(* PLC project prj, KAIST_DSLAB noNameNow 1, author bwkim *)
(* stored: creationDateTime 2017-1-22T00:06:53, modificationDateTime 2017-1-22T00:06:55 *)

PROGRAM Program1____sub1
  VAR
    SELECTION : INT;
  END_VAR
  VAR_INPUT
    CLKIO_ABOX_UAIF0 : INT;
  END_VAR
  VAR_INPUT
    CLKIO_ABOX_UAIF1 : INT;
  END_VAR
  VAR_INPUT
    CLKIO_ABOX_UAIF2 : INT;
  END_VAR
  VAR_INPUT
    CLKIO_ABOX_UAIF3 : INT;
  END_VAR
  VAR_INPUT
    CLKIO_ABoX_UAIF4 : INT;
  END_VAR
  VAR_INPUT
    FIN : INT;
  END_VAR
  VAR_INPUT
    FINN : INT;
  END_VAR
  VAR_INPUT
    OSCCLK_ABOX : INT;
  END_VAR
  VAR_OUTPUT
    ABOX_DAR : INT;
  END_VAR
  VAR_OUTPUT
    ACLKM_BTM_ABOX : INT;
  END_VAR
  VAR_OUTPUT
    ACLKS_PERI_AXI_AS : INT;
  END_VAR
  VAR_OUTPUT
    ACLK_ABOX_TOP : INT;
  END_VAR
  VAR_OUTPUT
    ACLK_PMU_ABOX : INT;
  END_VAR
  VAR_OUTPUT
    ACLK_PPMU_ABOX : INT;
  END_VAR
  VAR_OUTPUT
    ACLK_SYSREG_ABOX : INT;
  END_VAR
  VAR_OUTPUT
    AUD_CODEC_MCLK_DFTMUX_ABOX : INT;
  END_VAR
  VAR_OUTPUT
    BCLK_DSIF_ABOX_TOP : INT;
  END_VAR
  VAR_OUTPUT
    BCLK_UAIF2_ABOX_TOP : INT;
  END_VAR
  VAR_OUTPUT
    BCLK_UAIF3_ABOX_TOP : INT;
  END_VAR
  VAR_OUTPUT
    BCLK_UAIF4_ABOX_TOP : INT;
  END_VAR
  VAR_OUTPUT
    BCLK_UAIF_ABOX_TOP : INT;
  END_VAR
  VAR_OUTPUT
    CCLK_ASB_ABOX_TOP : INT;
  END_VAR
  VAR_OUTPUT
    CCLK_CA7_ABOX_TOP : INT;
  END_VAR
  VAR_OUTPUT
    CLKCMU_ABOX_CPUBOX : INT;
  END_VAR
  VAR_OUTPUT
    CLK_AXI_US_32to12 : INT;
  END_VAR
  VAR_OUTPUT
    CLK_RSTnSYNC_ABOX_CPU : INT;
  END_VAR
  VAR_OUTPUT
    CLK_RSTnSYNC_CLK_ABOX_B : INT;
  END_VAR
  VAR_OUTPUT
    CLK_RSTnSYNC_CLK_ABOX_CPU : INT;
  END_VAR
  VAR_OUTPUT
    CLK_RSTnSYNC_CLK_ABOX_DMIC : INT;
  END_VAR
  VAR_OUTPUT
    CLK_RSTnSYNC_CLK_ABOX_DSIF : INT;
  END_VAR
  VAR_OUTPUT
    CLK_RSTnSYNC_CLK_ABOX_UAIF0 : INT;
  END_VAR
  VAR_OUTPUT
    CLK_RSTnSYNC_CLK_ABOX_UAIF1 : INT;
  END_VAR
  VAR_OUTPUT
    CLK_RSTnSYNC_CLK_ABOX_UAIF2 : INT;
  END_VAR
  VAR_OUTPUT
    CLK_RSTnSYNC_CLK_ABOX_UAIF3 : INT;
  END_VAR
  VAR_OUTPUT
    CLK_RSTnSYNC_CLK_ABOX_UAIF4 : INT;
  END_VAR
  VAR_OUTPUT
    CLK_TREX_ABOX : INT;
  END_VAR
  VAR_OUTPUT
    CLK_WDT_AB0xCP0 : INT;
  END_VAR
  VAR_OUTPUT
    DIV_CLK_ABOX_BUS : INT;
  END_VAR
  VAR_OUTPUT
    DIV_CLK_ABOX_DSIF : INT;
  END_VAR
  VAR_OUTPUT
    I_CLK_ABOX_CMU_ABOX : INT;
  END_VAR
  VAR_OUTPUT
    I_CLK_LHM_AXI_P_ABOX : INT;
  END_VAR
  VAR_OUTPUT
    I_CLK_PERI_AXI_AS : INT;
  END_VAR
  VAR_OUTPUT
    I_CLK_RSSTnSYNC_CLK_ABOX : INT;
  END_VAR
  VAR_OUTPUT
    I_PCLK_BTM_ABOX : INT;
  END_VAR
  VAR_OUTPUT
    MUX_CLK_ABOX_CPU : INT;
  END_VAR
  VAR_OUTPUT
    PCLK_GPIO_ABOX : INT;
  END_VAR
  VAR_OUTPUT
    PCLK_LHS_AXI_D_ABOX : INT;
  END_VAR
  VAR_OUTPUT
    PCLK_PERI_AXI_AS : INT;
  END_VAR
  VAR_OUTPUT
    PCLK_PPMU_ABOX : INT;
  END_VAR
  VAR_OUTPUT
    PCLK_SMMU_ABOX : INT;
  END_VAR
  VAR_OUTPUT
    PLL_AUD : INT;
  END_VAR
  VAR_OUTPUT
    RSTnSYNC_CLK_ABOOX_UAI : INT;
  END_VAR
  VAR  (* added by the conversion: wires and edge detectors of the diagram *)
    _MIN2_DINT18_OUT : INT;
    _DINT_TO_REAL84_OUT : REAL;
    _DINT_TO_REAL122_OUT : REAL;
    _DINT_TO_REAL29_OUT : REAL;
    _DINT_TO_REAL88_OUT : REAL;
    _DINT_TO_REAL67_OUT : REAL;
    _DINT_TO_REAL89_OUT : REAL;
    _DINT_TO_REAL90_OUT : REAL;
    _REAL_TO_DINT26_OUT : DINT;
    _REAL_TO_DINT34_OUT : DINT;
    _DINT_TO_REAL56_OUT : REAL;
    _DINT_TO_REAL72_OUT : REAL;
    _DINT_TO_REAL73_OUT : REAL;
    _DINT_TO_REAL74_OUT : REAL;
    _DINT_TO_REAL124_OUT : REAL;
    _DINT_TO_REAL75_OUT : REAL;
    _DINT_TO_REAL76_OUT : REAL;
  END_VAR

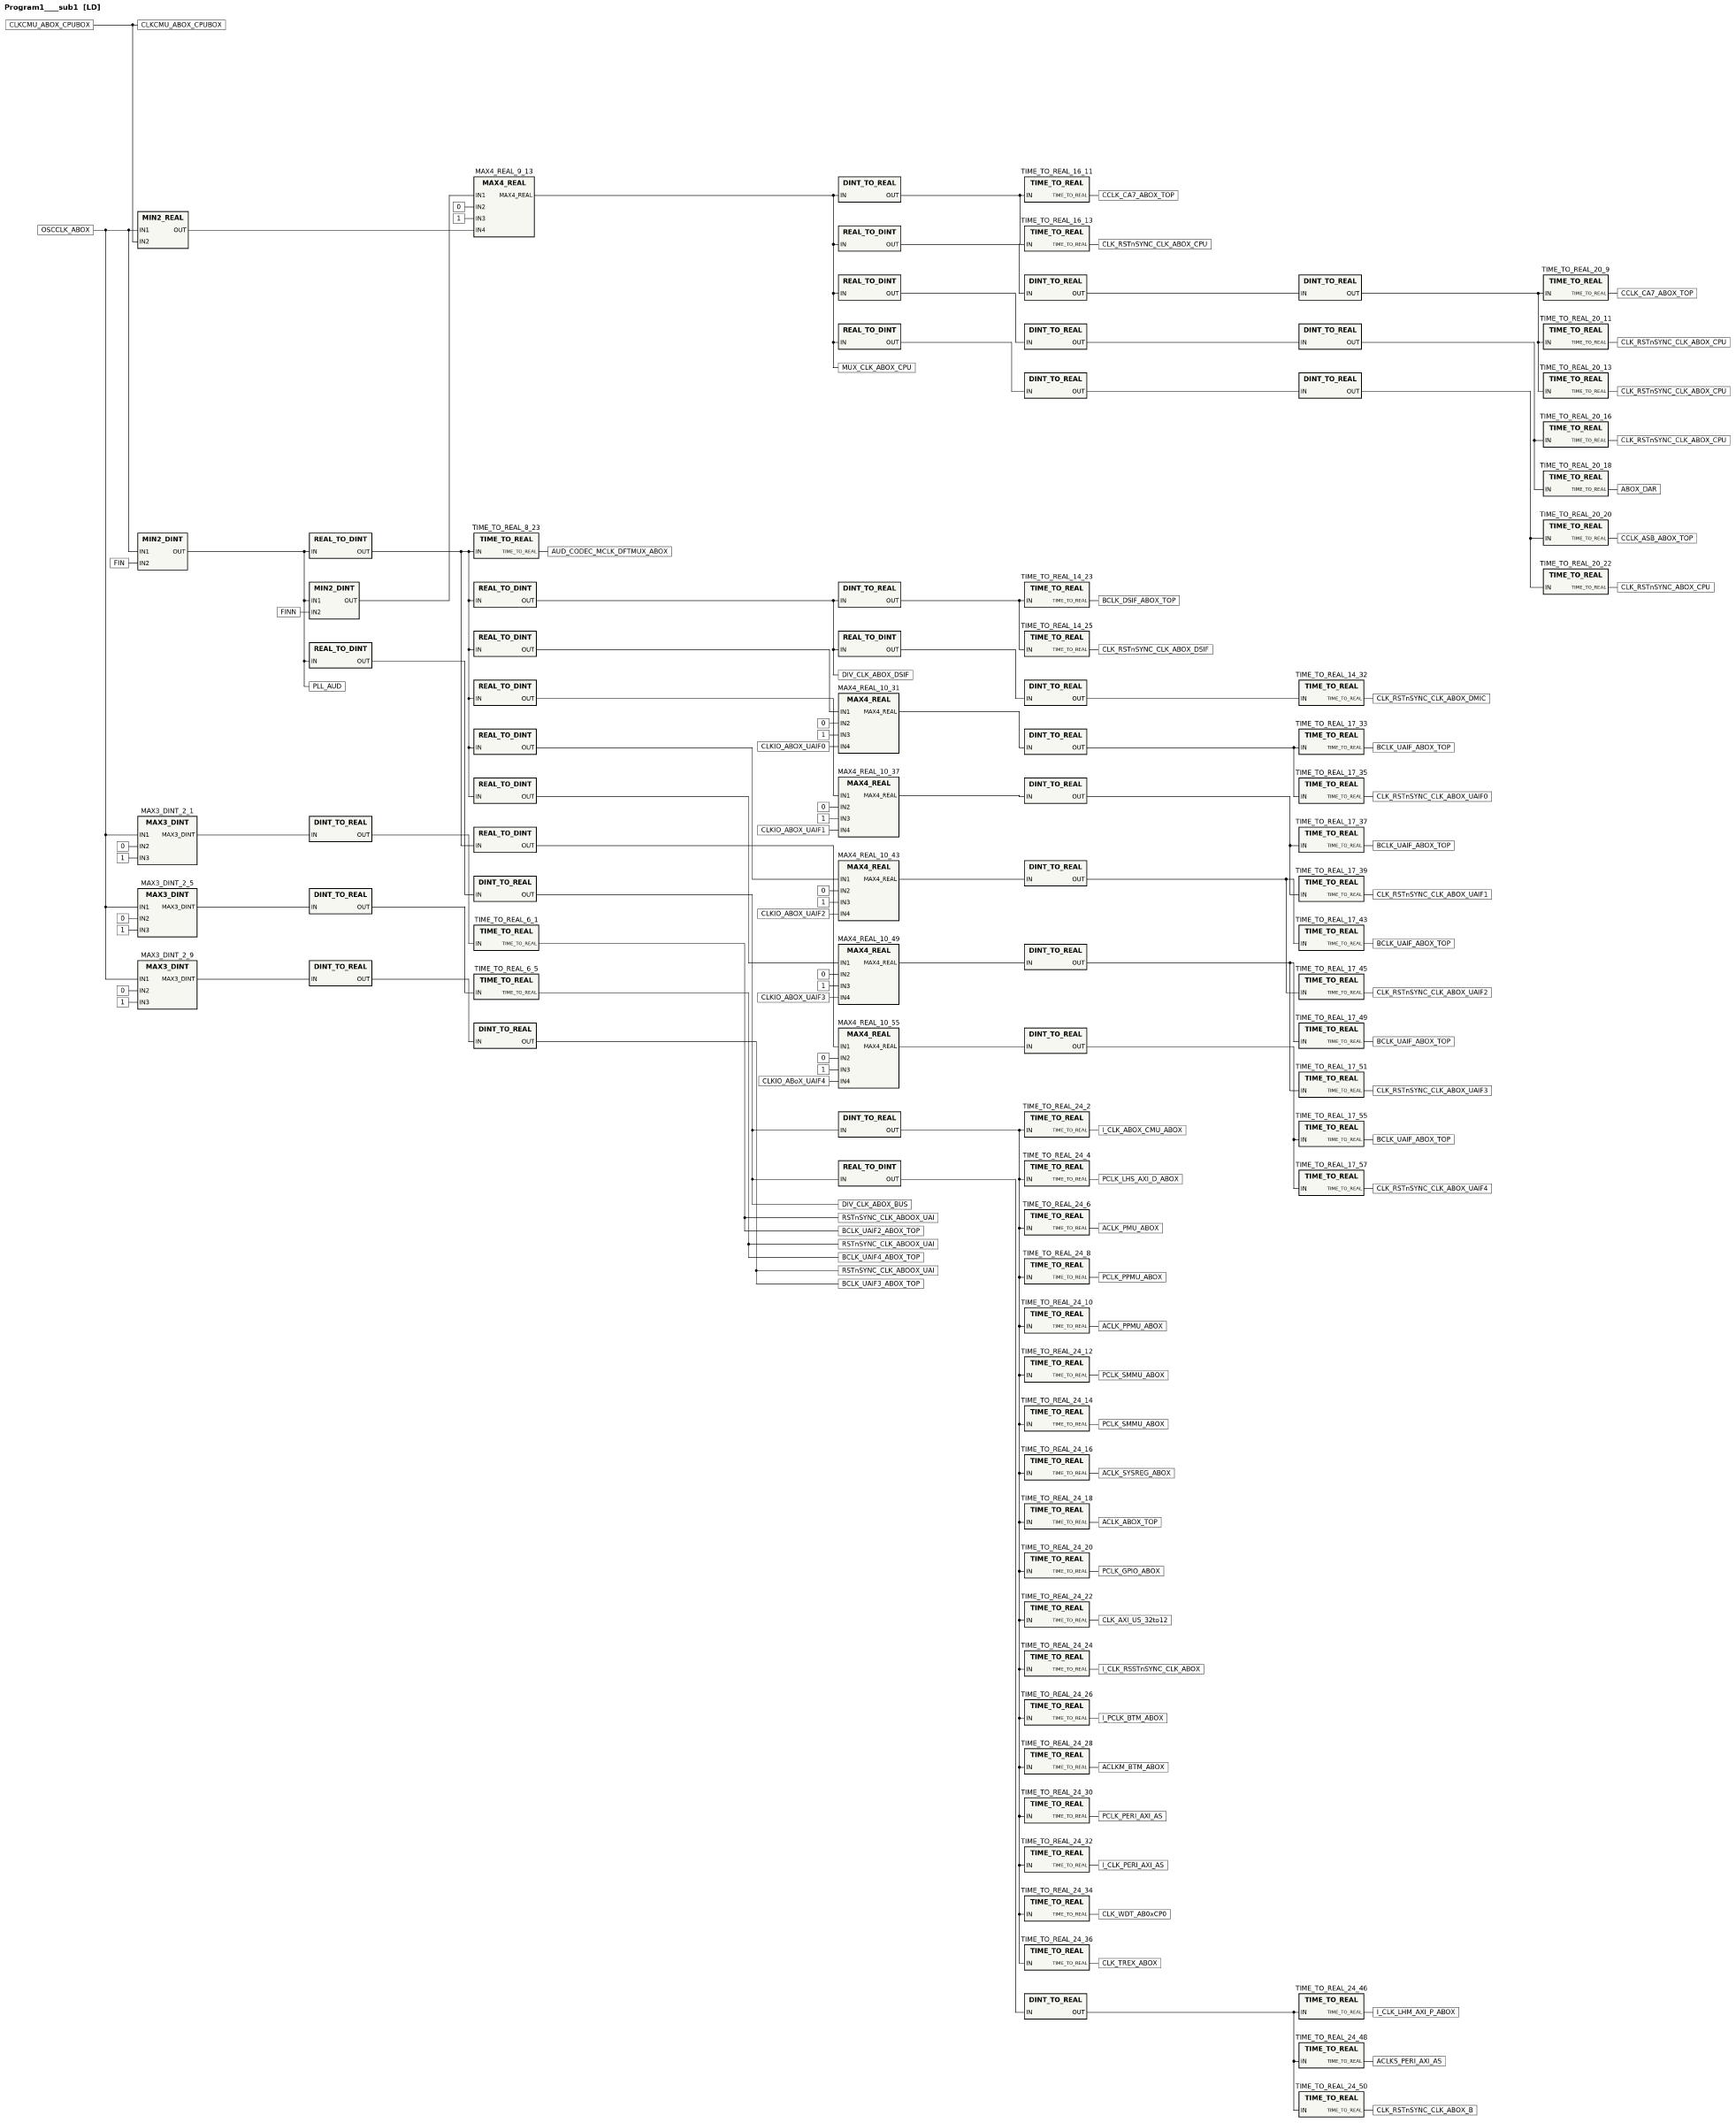
(* LD diagram, written out as Structured Text *)
MAX3_DINT_2_1(IN1 := OSCCLK_ABOX, IN2 := 0, IN3 := 1);
TIME_TO_REAL_6_1(IN := DINT_TO_REAL(MAX3_DINT_2_1.MAX3_DINT));
RSTnSYNC_CLK_ABOOX_UAI := TIME_TO_REAL_6_1.TIME_TO_REAL;
BCLK_UAIF2_ABOX_TOP := TIME_TO_REAL_6_1.TIME_TO_REAL;
_MIN2_DINT18_OUT := MIN2_DINT(OSCCLK_ABOX, FIN);
_DINT_TO_REAL84_OUT := DINT_TO_REAL(REAL_TO_DINT(_MIN2_DINT18_OUT));
_DINT_TO_REAL122_OUT := DINT_TO_REAL(_DINT_TO_REAL84_OUT);
TIME_TO_REAL_24_2(IN := _DINT_TO_REAL122_OUT);
I_CLK_ABOX_CMU_ABOX := TIME_TO_REAL_24_2.TIME_TO_REAL;
MAX3_DINT_2_5(IN1 := OSCCLK_ABOX, IN2 := 0, IN3 := 1);
TIME_TO_REAL_6_5(IN := DINT_TO_REAL(MAX3_DINT_2_5.MAX3_DINT));
RSTnSYNC_CLK_ABOOX_UAI := TIME_TO_REAL_6_5.TIME_TO_REAL;
TIME_TO_REAL_24_4(IN := _DINT_TO_REAL122_OUT);
PCLK_LHS_AXI_D_ABOX := TIME_TO_REAL_24_4.TIME_TO_REAL;
BCLK_UAIF4_ABOX_TOP := TIME_TO_REAL_6_5.TIME_TO_REAL;
TIME_TO_REAL_24_6(IN := _DINT_TO_REAL122_OUT);
ACLK_PMU_ABOX := TIME_TO_REAL_24_6.TIME_TO_REAL;
MAX3_DINT_2_9(IN1 := OSCCLK_ABOX, IN2 := 0, IN3 := 1);
_DINT_TO_REAL29_OUT := DINT_TO_REAL(DINT_TO_REAL(MAX3_DINT_2_9.MAX3_DINT));
RSTnSYNC_CLK_ABOOX_UAI := _DINT_TO_REAL29_OUT;
TIME_TO_REAL_24_8(IN := _DINT_TO_REAL122_OUT);
PCLK_PPMU_ABOX := TIME_TO_REAL_24_8.TIME_TO_REAL;
BCLK_UAIF3_ABOX_TOP := _DINT_TO_REAL29_OUT;
MAX4_REAL_9_13(IN1 := MIN2_DINT(_MIN2_DINT18_OUT, FINN), IN2 := 0, IN3 := 1, IN4 := MIN2_REAL(OSCCLK_ABOX, CLKCMU_ABOX_CPUBOX));
_DINT_TO_REAL88_OUT := DINT_TO_REAL(DINT_TO_REAL(REAL_TO_DINT(MAX4_REAL_9_13.MAX4_REAL)));
TIME_TO_REAL_20_9(IN := _DINT_TO_REAL88_OUT);
CCLK_CA7_ABOX_TOP := TIME_TO_REAL_20_9.TIME_TO_REAL;
TIME_TO_REAL_24_10(IN := _DINT_TO_REAL122_OUT);
ACLK_PPMU_ABOX := TIME_TO_REAL_24_10.TIME_TO_REAL;
MUX_CLK_ABOX_CPU := MAX4_REAL_9_13.MAX4_REAL;
_DINT_TO_REAL67_OUT := DINT_TO_REAL(MAX4_REAL_9_13.MAX4_REAL);
TIME_TO_REAL_16_11(IN := _DINT_TO_REAL67_OUT);
CCLK_CA7_ABOX_TOP := TIME_TO_REAL_16_11.TIME_TO_REAL;
TIME_TO_REAL_20_11(IN := _DINT_TO_REAL88_OUT);
CLK_RSTnSYNC_CLK_ABOX_CPU := TIME_TO_REAL_20_11.TIME_TO_REAL;
PLL_AUD := _MIN2_DINT18_OUT;
TIME_TO_REAL_24_12(IN := _DINT_TO_REAL122_OUT);
PCLK_SMMU_ABOX := TIME_TO_REAL_24_12.TIME_TO_REAL;
TIME_TO_REAL_16_13(IN := _DINT_TO_REAL67_OUT);
CLK_RSTnSYNC_CLK_ABOX_CPU := TIME_TO_REAL_16_13.TIME_TO_REAL;
TIME_TO_REAL_20_13(IN := _DINT_TO_REAL88_OUT);
CLK_RSTnSYNC_CLK_ABOX_CPU := TIME_TO_REAL_20_13.TIME_TO_REAL;
TIME_TO_REAL_24_14(IN := _DINT_TO_REAL122_OUT);
PCLK_SMMU_ABOX := TIME_TO_REAL_24_14.TIME_TO_REAL;
_DINT_TO_REAL89_OUT := DINT_TO_REAL(DINT_TO_REAL(REAL_TO_DINT(MAX4_REAL_9_13.MAX4_REAL)));
TIME_TO_REAL_20_16(IN := _DINT_TO_REAL89_OUT);
CLK_RSTnSYNC_CLK_ABOX_CPU := TIME_TO_REAL_20_16.TIME_TO_REAL;
TIME_TO_REAL_24_16(IN := _DINT_TO_REAL122_OUT);
ACLK_SYSREG_ABOX := TIME_TO_REAL_24_16.TIME_TO_REAL;
TIME_TO_REAL_20_18(IN := _DINT_TO_REAL89_OUT);
ABOX_DAR := TIME_TO_REAL_20_18.TIME_TO_REAL;
TIME_TO_REAL_24_18(IN := _DINT_TO_REAL122_OUT);
ACLK_ABOX_TOP := TIME_TO_REAL_24_18.TIME_TO_REAL;
CLKCMU_ABOX_CPUBOX := CLKCMU_ABOX_CPUBOX;
_DINT_TO_REAL90_OUT := DINT_TO_REAL(DINT_TO_REAL(REAL_TO_DINT(MAX4_REAL_9_13.MAX4_REAL)));
TIME_TO_REAL_20_20(IN := _DINT_TO_REAL90_OUT);
CCLK_ASB_ABOX_TOP := TIME_TO_REAL_20_20.TIME_TO_REAL;
TIME_TO_REAL_24_20(IN := _DINT_TO_REAL122_OUT);
PCLK_GPIO_ABOX := TIME_TO_REAL_24_20.TIME_TO_REAL;
_REAL_TO_DINT26_OUT := REAL_TO_DINT(_MIN2_DINT18_OUT);
_REAL_TO_DINT34_OUT := REAL_TO_DINT(_REAL_TO_DINT26_OUT);
DIV_CLK_ABOX_DSIF := _REAL_TO_DINT34_OUT;
TIME_TO_REAL_20_22(IN := _DINT_TO_REAL90_OUT);
CLK_RSTnSYNC_ABOX_CPU := TIME_TO_REAL_20_22.TIME_TO_REAL;
TIME_TO_REAL_24_22(IN := _DINT_TO_REAL122_OUT);
CLK_AXI_US_32to12 := TIME_TO_REAL_24_22.TIME_TO_REAL;
TIME_TO_REAL_8_23(IN := _REAL_TO_DINT26_OUT);
AUD_CODEC_MCLK_DFTMUX_ABOX := TIME_TO_REAL_8_23.TIME_TO_REAL;
_DINT_TO_REAL56_OUT := DINT_TO_REAL(_REAL_TO_DINT34_OUT);
TIME_TO_REAL_14_23(IN := _DINT_TO_REAL56_OUT);
BCLK_DSIF_ABOX_TOP := TIME_TO_REAL_14_23.TIME_TO_REAL;
DIV_CLK_ABOX_BUS := _DINT_TO_REAL84_OUT;
TIME_TO_REAL_24_24(IN := _DINT_TO_REAL122_OUT);
I_CLK_RSSTnSYNC_CLK_ABOX := TIME_TO_REAL_24_24.TIME_TO_REAL;
TIME_TO_REAL_14_25(IN := _DINT_TO_REAL56_OUT);
CLK_RSTnSYNC_CLK_ABOX_DSIF := TIME_TO_REAL_14_25.TIME_TO_REAL;
TIME_TO_REAL_24_26(IN := _DINT_TO_REAL122_OUT);
I_PCLK_BTM_ABOX := TIME_TO_REAL_24_26.TIME_TO_REAL;
TIME_TO_REAL_24_28(IN := _DINT_TO_REAL122_OUT);
ACLKM_BTM_ABOX := TIME_TO_REAL_24_28.TIME_TO_REAL;
TIME_TO_REAL_24_30(IN := _DINT_TO_REAL122_OUT);
PCLK_PERI_AXI_AS := TIME_TO_REAL_24_30.TIME_TO_REAL;
TIME_TO_REAL_14_32(IN := DINT_TO_REAL(REAL_TO_DINT(_REAL_TO_DINT34_OUT)));
CLK_RSTnSYNC_CLK_ABOX_DMIC := TIME_TO_REAL_14_32.TIME_TO_REAL;
TIME_TO_REAL_24_32(IN := _DINT_TO_REAL122_OUT);
I_CLK_PERI_AXI_AS := TIME_TO_REAL_24_32.TIME_TO_REAL;
MAX4_REAL_10_31(IN1 := REAL_TO_DINT(_REAL_TO_DINT26_OUT), IN2 := 0, IN3 := 1, IN4 := CLKIO_ABOX_UAIF0);
_DINT_TO_REAL72_OUT := DINT_TO_REAL(MAX4_REAL_10_31.MAX4_REAL);
TIME_TO_REAL_17_33(IN := _DINT_TO_REAL72_OUT);
BCLK_UAIF_ABOX_TOP := TIME_TO_REAL_17_33.TIME_TO_REAL;
TIME_TO_REAL_24_34(IN := _DINT_TO_REAL122_OUT);
CLK_WDT_AB0xCP0 := TIME_TO_REAL_24_34.TIME_TO_REAL;
TIME_TO_REAL_17_35(IN := _DINT_TO_REAL72_OUT);
CLK_RSTnSYNC_CLK_ABOX_UAIF0 := TIME_TO_REAL_17_35.TIME_TO_REAL;
TIME_TO_REAL_24_36(IN := _DINT_TO_REAL122_OUT);
CLK_TREX_ABOX := TIME_TO_REAL_24_36.TIME_TO_REAL;
MAX4_REAL_10_37(IN1 := REAL_TO_DINT(_REAL_TO_DINT26_OUT), IN2 := 0, IN3 := 1, IN4 := CLKIO_ABOX_UAIF1);
_DINT_TO_REAL73_OUT := DINT_TO_REAL(MAX4_REAL_10_37.MAX4_REAL);
TIME_TO_REAL_17_37(IN := _DINT_TO_REAL73_OUT);
BCLK_UAIF_ABOX_TOP := TIME_TO_REAL_17_37.TIME_TO_REAL;
TIME_TO_REAL_17_39(IN := _DINT_TO_REAL73_OUT);
CLK_RSTnSYNC_CLK_ABOX_UAIF1 := TIME_TO_REAL_17_39.TIME_TO_REAL;
MAX4_REAL_10_43(IN1 := REAL_TO_DINT(_REAL_TO_DINT26_OUT), IN2 := 0, IN3 := 1, IN4 := CLKIO_ABOX_UAIF2);
_DINT_TO_REAL74_OUT := DINT_TO_REAL(MAX4_REAL_10_43.MAX4_REAL);
TIME_TO_REAL_17_43(IN := _DINT_TO_REAL74_OUT);
BCLK_UAIF_ABOX_TOP := TIME_TO_REAL_17_43.TIME_TO_REAL;
TIME_TO_REAL_17_45(IN := _DINT_TO_REAL74_OUT);
CLK_RSTnSYNC_CLK_ABOX_UAIF2 := TIME_TO_REAL_17_45.TIME_TO_REAL;
_DINT_TO_REAL124_OUT := DINT_TO_REAL(REAL_TO_DINT(_DINT_TO_REAL84_OUT));
TIME_TO_REAL_24_46(IN := _DINT_TO_REAL124_OUT);
I_CLK_LHM_AXI_P_ABOX := TIME_TO_REAL_24_46.TIME_TO_REAL;
TIME_TO_REAL_24_48(IN := _DINT_TO_REAL124_OUT);
ACLKS_PERI_AXI_AS := TIME_TO_REAL_24_48.TIME_TO_REAL;
MAX4_REAL_10_49(IN1 := REAL_TO_DINT(_REAL_TO_DINT26_OUT), IN2 := 0, IN3 := 1, IN4 := CLKIO_ABOX_UAIF3);
_DINT_TO_REAL75_OUT := DINT_TO_REAL(MAX4_REAL_10_49.MAX4_REAL);
TIME_TO_REAL_17_49(IN := _DINT_TO_REAL75_OUT);
BCLK_UAIF_ABOX_TOP := TIME_TO_REAL_17_49.TIME_TO_REAL;
TIME_TO_REAL_24_50(IN := _DINT_TO_REAL124_OUT);
CLK_RSTnSYNC_CLK_ABOX_B := TIME_TO_REAL_24_50.TIME_TO_REAL;
TIME_TO_REAL_17_51(IN := _DINT_TO_REAL75_OUT);
CLK_RSTnSYNC_CLK_ABOX_UAIF3 := TIME_TO_REAL_17_51.TIME_TO_REAL;
MAX4_REAL_10_55(IN1 := REAL_TO_DINT(_REAL_TO_DINT26_OUT), IN2 := 0, IN3 := 1, IN4 := CLKIO_ABoX_UAIF4);
_DINT_TO_REAL76_OUT := DINT_TO_REAL(MAX4_REAL_10_55.MAX4_REAL);
TIME_TO_REAL_17_55(IN := _DINT_TO_REAL76_OUT);
BCLK_UAIF_ABOX_TOP := TIME_TO_REAL_17_55.TIME_TO_REAL;
TIME_TO_REAL_17_57(IN := _DINT_TO_REAL76_OUT);
CLK_RSTnSYNC_CLK_ABOX_UAIF4 := TIME_TO_REAL_17_57.TIME_TO_REAL;
END_PROGRAM
